FUNCTION_BLOCK E_SPLIT_5 (* Composite Function Block Type *)
  (* Standard: 61499-2 *)
  (* Version 0.0, 2018-11-02, 4DIAC-IDE, 4DIAC-Consortium *)
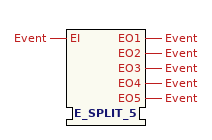
  EVENT_INPUT
    EI;
  END_EVENT
  EVENT_OUTPUT
    EO1;
    EO2;
    EO3;
    EO4;
    EO5;
  END_EVENT
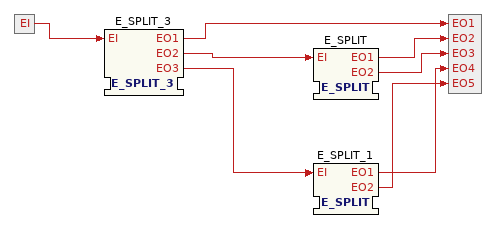
  FBS
    E_SPLIT_3 : E_SPLIT_3;
    E_SPLIT : E_SPLIT;
    E_SPLIT_1 : E_SPLIT;
  END_FBS
  EVENT_CONNECTIONS
    EI TO E_SPLIT_3.EI;
    E_SPLIT_3.EO1 TO EO1;
    E_SPLIT_3.EO2 TO E_SPLIT.EI;
    E_SPLIT.EO1 TO EO2;
    E_SPLIT.EO2 TO EO3;
    E_SPLIT_3.EO3 TO E_SPLIT_1.EI;
    E_SPLIT_1.EO1 TO EO4;
    E_SPLIT_1.EO2 TO EO5;
  END_CONNECTIONS
END_FUNCTION_BLOCK
